TYPE (* logiBUS_DI Struct *)
  (* Version 1.0, 2025-07-21, franz *)
  PACKAGE logiBUS::io::AI;
  logiBUS_AI_S : STRUCT
    Pin : USINT := 255;
  END_STRUCT;
END_TYPE
